TYPE stUNbase :
STRUCT
	sTagName : STRING;
	sDescription : STRING;
END_STRUCT
END_TYPE

(* stored: Version 1.1.0.1, ProductVersion 3.1.4024.12
   DUT stUNbase: Id {08ed44d5-5094-4f84-9297-f1f05b2700a2} *)
